# EPICS autosave request: ADPSL/iocs/pslIOC/iocBoot/iocPSL/auto_settings.req
file "PSL_settings.req",          P=$(P),  R=cam1:
file "NDFile_settings.req",       P=$(P),  R=cam1:
file "NDStdArrays_settings.req",  P=$(P),  R=image1:
file "commonPlugin_settings.req", P=$(P)
